SUBAPPLICATION Uebung_083_AX (* Beispiel für AUDI_CTUD_UDINT (Adapter-basiert) *)
  (* Standard: 61499-2; Description: Copyright (c) 2023 Meisterschulen am Ostbahnhof This program and the accompanying materials are made available under the terms of the Eclipse Public License 2.0 which is available at https://www.eclipse.org/legal/epl-2.0/ SPDX-License-Identifier: EPL-2.0 *)
  (* Version 1.0, 2026-01-17, Franz Höpfinger, Meisterschulen am Ostbahnhof, initial API and implementation and/or initial documentation *)
  PACKAGE Uebungen;
  IMPORT Uebungen::const::UT::DefaultPool::OutputNumber_N1;
  IMPORT logiBUS::io::DI::logiBUS_DI::Input_I1;
  IMPORT logiBUS::io::DI::logiBUS_DI::Input_I2;
  IMPORT logiBUS::io::DI::logiBUS_DI::Input_I3;
  IMPORT logiBUS::io::DI::logiBUS_DI::Input_I4;
  IMPORT logiBUS::io::DI::logiBUS_DI_Events::BUTTON_SINGLE_CLICK;
  IMPORT logiBUS::io::DQ::logiBUS_DO::Output_Q1;
  IMPORT logiBUS::io::DQ::logiBUS_DO::Output_Q2;
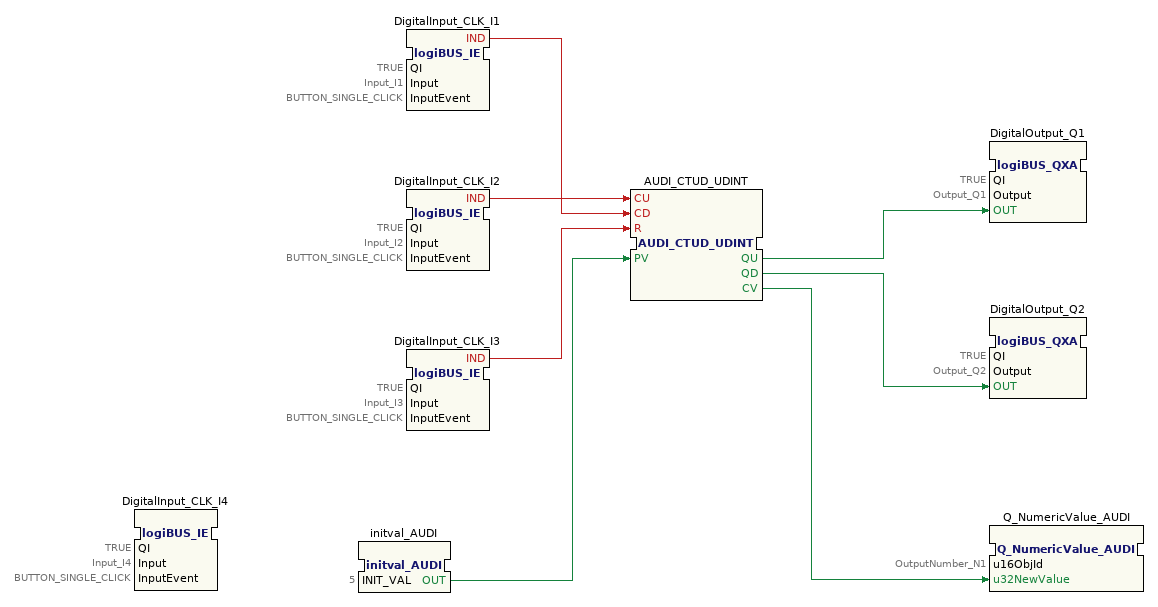
  FBS
    DigitalOutput_Q1 : logiBUS::io::DQ::logiBUS_QXA(QI := TRUE, Output := Output_Q1);
    DigitalInput_CLK_I1 : logiBUS::io::DI::logiBUS_IE(QI := TRUE, Input := Input_I1, InputEvent := BUTTON_SINGLE_CLICK);
    AUDI_CTUD_UDINT : adapter::events::unidirectional::AUDI_CTUD_UDINT;
    DigitalInput_CLK_I2 : logiBUS::io::DI::logiBUS_IE(QI := TRUE, Input := Input_I2, InputEvent := BUTTON_SINGLE_CLICK);
    DigitalInput_CLK_I3 : logiBUS::io::DI::logiBUS_IE(QI := TRUE, Input := Input_I3, InputEvent := BUTTON_SINGLE_CLICK);
    DigitalInput_CLK_I4 : logiBUS::io::DI::logiBUS_IE(QI := TRUE, Input := Input_I4, InputEvent := BUTTON_SINGLE_CLICK);
    DigitalOutput_Q2 : logiBUS::io::DQ::logiBUS_QXA(QI := TRUE, Output := Output_Q2);
    Q_NumericValue_AUDI : isobus::UT::Q::Q_NumericValue_AUDI(u16ObjId := OutputNumber_N1);
    initval_AUDI : adapter::types::unidirectional::AUDI::initval::initval_AUDI(INIT_VAL := 5);
  END_FBS
  EVENT_CONNECTIONS
    DigitalInput_CLK_I1.IND TO AUDI_CTUD_UDINT.CU;
    DigitalInput_CLK_I2.IND TO AUDI_CTUD_UDINT.CD;
    DigitalInput_CLK_I3.IND TO AUDI_CTUD_UDINT.R;
  END_CONNECTIONS
  ADAPTER_CONNECTIONS
    AUDI_CTUD_UDINT.QU TO DigitalOutput_Q1.OUT;
    AUDI_CTUD_UDINT.QD TO DigitalOutput_Q2.OUT;
    AUDI_CTUD_UDINT.CV TO Q_NumericValue_AUDI.u32NewValue;
    initval_AUDI.OUT TO AUDI_CTUD_UDINT.PV;
  END_CONNECTIONS
END_SUBAPPLICATION
